FUNCTION_BLOCK SM_LineRegulator EXTENDS StateMachine
VAR_INPUT
	 sSubscription1 : STRING(8);
	 sSubscription2 : STRING(8);
	 sSubscription3 : STRING(8);
END_VAR
VAR_OUTPUT
END_VAR
VAR
	fbTurntable : Turntable;

	aRollerConveyors : ARRAY[1..3] OF RollerConveyor;
	fbRollerConveyorExit : RollerConveyor;
	fbReadyStepWorker : FB_StepWorker;
	fbBusyStepWorker : FB_StepWorker;
	fbInitStepWorker : FB_StepWorker;
	
	messageIndex : UINT;
	stMqttPayload : ST_MqttPayload;
	aSubscriptions : ARRAY[1..3] OF STRING(8);
	uiSubscriptionsCycler : UINT := 1;
END_VAR

SUPER^();
fbTurntable();
aRollerConveyors[1]();
aRollerConveyors[3]();

METHOD PROTECTED   Busy : BOOL
VAR_INPUT
END_VAR
fbBusyStepWorker();
CASE fbBusyStepWorker.uiStep OF

	0:
	
		aRollerConveyors[uiSubscriptionsCycler].On();
		CASE uiSubscriptionsCycler OF
		
			1:
				fbTurntable.RollMinus();
				fbTurntable.Turn();
			
			2:
				fbTurntable.RollPlus();
			
			3:
				fbTurntable.RollPlus();
				fbTurntable.Turn();
		END_CASE
		
		fbBusyStepWorker
			.mAddCondition(itfStepCondition := fbTurntable.fbBackLimit.getSignal)
			.mNextStep(10);
			
	10:
	
		aRollerConveyors[uiSubscriptionsCycler].Off();
		CASE uiSubscriptionsCycler OF
		
			1:
				fbTurntable.StopRolling();			
				fbTurntable.UnTurn();
				fbBusyStepWorker
					.mSetTimer(T#2S)
					.mNextStep(20);
			
			2:
				fbBusyStepWorker.mNextStep(30);
			
			3:
				fbTurntable.StopRolling();
				fbTurntable.UnTurn();
				fbBusyStepWorker
					.mSetTimer(T#2S)
					.mNextStep(20);
		END_CASE
		
	20:
	
		fbTurntable.RollPlus();
		fbRollerConveyorExit.On();
		fbBusyStepWorker
			.mSetTimer(T#10S)
			.mNextStep(30);
	30:	
	
		IF NOT fbTurntable.fbBackLimit.bSignal
			AND NOT fbTurntable.fbFrontLimit.bSignal
		THEN
			fbRollerConveyorExit.Off();
			fbBusyStepWorker
				.mSetTimer(T#1S)
				.mNextStep(40);
		END_IF
		
	40:
	
		fbBusyStepWorker.mNextStep(0);
		Done();
		
	
END_CASE
END_METHOD

METHOD PROTECTED  Error : BOOL
VAR_INPUT
END_VAR
END_METHOD

METHOD PROTECTED  Idle : BOOL
VAR_INPUT
END_VAR
END_METHOD

METHOD PROTECTED  Init : BOOL
VAR_INPUT
END_VAR
fbInitStepWorker();
CASE fbInitStepWorker.uiStep OF

	0: 
	
		IF ADS.fbAdsConnector.isConnected
		THEN
			fbInitStepWorker.mNextStep(10);
		END_IF
		
	10:
	
		IF ADS.fbMqttClient.Subscribe(sSubscription1)
		THEN			
			fbInitStepWorker.mNextStep(20);
		END_IF
		
	20:
	
		IF ADS.fbMqttClient.Subscribe(sSubscription2)
		THEN			
			fbInitStepWorker.mNextStep(30);
		END_IF
		
	30:
		
		IF ADS.fbMqttClient.Subscribe(sSubscription3)
		THEN		
			aSubscriptions[1] := sSubscription1;
			aSubscriptions[2] := sSubscription2;
			aSubscriptions[3] := sSubscription3;
			Start();
		END_IF		
		
END_CASE
END_METHOD

METHOD PROTECTED  Prepare : BOOL
VAR_INPUT
END_VAR
END_METHOD

METHOD PROTECTED  Ready : BOOL
VAR_INPUT
END_VAR
VAR
	
END_VAR
fbReadyStepWorker();


CASE fbReadyStepWorker.uiStep OF

	0: 
		IF NOT fbTurntable.bBackLimit
			AND NOT fbTurntable.bFrontLimit
		THEN
			fbReadyStepWorker.mNextStep(10);
		END_IF
		
	10:
	
		IF uiSubscriptionsCycler = 3
		THEN
			uiSubscriptionsCycler := 1;
		ELSE
			uiSubscriptionsCycler := uiSubscriptionsCycler + 1;
		END_IF
		
		messageIndex := ADS.fbMqttClient.isNewMessage(aSubscriptions[uiSubscriptionsCycler]);
		IF messageIndex > 0
		THEN
			stMqttPayload := Ads.fbMqttClient.getNewMessage(messageIndex);
			fbReadyStepWorker.mNextStep(20);
		END_IF
		
	20:	
		Ads.fbMqttClient.Publish(aSubscriptions[uiSubscriptionsCycler],stMqttPayload);
		fbReadyStepWorker.mNextStep(0);
		Execute();
		
END_CASE
END_METHOD

METHOD PROTECTED  Waiting : BOOL
VAR_INPUT
END_VAR
END_METHOD

END_FUNCTION_BLOCK

(* stored: Version 1.1.0.1, ProductVersion 3.1.4024.2
   POU SM_LineRegulator: Id {ad4b4131-efe4-4f92-890f-d8bb1cb3f800}, SpecialFunc None
   Method Busy: Id {bacf8a3e-55e0-476f-ae74-184212c7d4f8}
   Method Error: Id {96ce5d74-7a3f-42d7-b0d0-3590a804dfe2}
   Method Idle: Id {38cba348-d9fd-409a-9b9e-4554d87a396f}
   Method Init: Id {f1a298c1-d662-4861-a48d-11d144d0f0c6}
   Method Prepare: Id {1f0fec7d-c33b-4175-960e-d20abfbb4fbd}
   Method Ready: Id {b00cb338-3e9d-4791-9660-cd67b71e4703}
   Method Waiting: Id {f685a573-862a-4fe6-a9e9-e1ec45aadb97} *)
